TYPE
	NW_BUF_LONG  : ARRAY[0..NETWORK_BUFFER_LONG_SIZE] OF BYTE;
END_TYPE

(* stored: Version 1.1.0.1, ProductVersion 3.1.4024.4
   DUT NW_BUF_LONG: Id {9395f7dd-59af-4e3f-bb13-e118edf120de} *)
